// TIA Portal V19 export
DATA_BLOCK "Alarms_DB"   // DB2
// stored: InstanceOfName Alarms, InstanceOfType FB
"Alarms"
BEGIN
END_DATA_BLOCK
